(* IEC 61131-3 sources: POMIRTS_lab3/AS/Library_2/AsNxCoM, 3 files *)

(* ---- AsNxCoM.typ ---- *)
TYPE
	nxcomEmcyTelegram_t		: STRUCT			(*emergency telegram*)
		data				: ARRAY[0..7] OF USINT;
	END_STRUCT;

	nxcomEmcyTelegrams_t	: STRUCT			(*array of emergency telegrams*)
		telegram			: ARRAY[0..4] OF nxcomEmcyTelegram_t;
	END_STRUCT;
END_TYPE

(* ---- AsNxCoM.fun ---- *)
{REDUND_CONTEXT} {REDUND_UNREPLICABLE} FUNCTION_BLOCK nxcomGetState			(*get state*)
	VAR_INPUT
		enable			: BOOL;			(*enables execution*)
		pDevice			: UDINT;		(*interface name given as a pointer, e.g., "SL<x>.SS<y>.IF<z>"*)
		node			: USINT;		(*node id*)
		flags			: UDINT;		(*flags*)
	END_VAR
	VAR
        _state			: UINT;			(*internal variable*)
		_result			: UINT;			(*internal variable*)
        _srcId			: UDINT;		(*internal variable*)
	END_VAR
	VAR_OUTPUT
		status			: UINT;			(*execution status: ERR_OK, ERR_FUB_ENABLE_FALSE, ERR_FUB_BUSY, 0xXXXX = see help*)
		coStatus		: UDINT;		(*CANopen stack status*)
		nmtState		: UDINT;		(*state*)
	END_VAR
END_FUNCTION_BLOCK

{REDUND_CONTEXT} {REDUND_UNREPLICABLE} FUNCTION_BLOCK nxcomRecvEmcyDev			(*receive emergency telegrams*)
	VAR_INPUT
		enable			: BOOL;			(*enables execution*)
		pDevice			: UDINT;		(*interface name given as a pointer, e.g., "SL<x>.SS<y>.IF<z>"*)
		node			: USINT;		(*node id*)
		flags			: UDINT;		(*flags*)
		pEmcyData		: UDINT;		(*data field for emergency entries given as pointer (consisting of 5 blocks each sized 8 bytes)*)
	END_VAR
	VAR
        _state			: UINT;			(*internal variable*)
		_result			: UINT;			(*internal variable*)
        _srcId			: UDINT;		(*internal variable*)
	END_VAR
	VAR_OUTPUT
		status			: UINT;			(*execution status: ERR_OK, ERR_FUB_ENABLE_FALSE, ERR_FUB_BUSY, 0xXXXX = see help*)
		coStatus		: UDINT;		(*CANopen stack status*)
		emcyCount		: UDINT;		(*current number of emergency telegrams in buffer*)
	END_VAR
END_FUNCTION_BLOCK

{REDUND_CONTEXT} {REDUND_UNREPLICABLE} FUNCTION_BLOCK nxcomGetDiag				(*get node diagnostics*)
	VAR_INPUT
		enable			: BOOL;			(*enables execution*)
		pDevice			: UDINT;		(*interface name given as a pointer, e.g., "SL<x>.SS<y>.IF<z>"*)
		node			: USINT;		(*node id*)
		flags			: UDINT;		(*flags*)
		pEmcyData		: UDINT;		(*data field for emergency entries given as pointer (consisting of 5 blocks each sized 8 bytes)*)
	END_VAR
	VAR
        _state			: UINT;			(*internal variable*)
		_result			: UINT;			(*internal variable*)
        _srcId			: UDINT;		(*internal variable*)
	END_VAR
	VAR_OUTPUT
		status			: UINT;			(*execution status: ERR_OK, ERR_FUB_ENABLE_FALSE, ERR_FUB_BUSY, 0xXXXX = see help*)
		coStatus		: UDINT;		(*CANopen stack status*)
		nodeFlags		: UDINT;		(*node flags*)
		lastDiagInfo	: UDINT;		(*last diagnostics info*)
		devTypeValid	: BOOL;			(*is device type valid*)
		devType			: UDINT;		(*device type*)
		nmtState		: UDINT;		(*nmt state*)
		emcyCount		: UDINT;		(*current number of emergency telegrams in buffer*)
		addInfo			: UDINT;		(*additional info*)
	END_VAR
END_FUNCTION_BLOCK

{REDUND_CONTEXT} {REDUND_UNREPLICABLE} FUNCTION_BLOCK nxcomNmt					(*send NMT command*)
	VAR_INPUT
		enable			: BOOL;			(*enables execution*)
		pDevice			: UDINT;		(*interface name given as a pointer, e.g., "SL<x>.SS<y>.IF<z>"*)
		node			: USINT;		(*node id*)
		command			: UDINT;		(*NMT command*)
	END_VAR
	VAR
        _state			: UINT;			(*internal variable*)
		_result			: UINT;			(*internal variable*)
        _srcId			: UDINT;		(*internal variable*)
	END_VAR
	VAR_OUTPUT
		status			: UINT;			(*execution status: ERR_OK, ERR_FUB_ENABLE_FALSE, ERR_FUB_BUSY, 0xXXXX = see help*)
		coStatus		: UDINT;		(*CANopen stack status*)
	END_VAR
END_FUNCTION_BLOCK

{REDUND_CONTEXT} {REDUND_UNREPLICABLE} FUNCTION_BLOCK nxcomSdoRead				(*read SDO data*)
	VAR_INPUT
		enable			: BOOL;			(*enables execution*)
		pDevice			: UDINT;		(*interface name given as a pointer, e.g., "SL<x>.SS<y>.IF<z>"*)
		node			: USINT;		(*node id*)
		index			: UDINT;		(*index*)
		subIndex		: UDINT;		(*sub index*)
		dataCount		: UDINT;		(*data count*)
		pData			: UDINT;		(*sdo data given as pointer*)
	END_VAR
	VAR
        _state			: UINT;			(*internal variable*)
		_result			: UINT;			(*internal variable*)
        _srcId			: UDINT;		(*internal variable*)
	END_VAR
	VAR_OUTPUT
		status			: UINT;			(*execution status: ERR_OK, ERR_FUB_ENABLE_FALSE, ERR_FUB_BUSY, 0xXXXX = see help*)
		coStatus		: UDINT;		(*CANopen stack status*)
	END_VAR
END_FUNCTION_BLOCK

{REDUND_CONTEXT} {REDUND_UNREPLICABLE} FUNCTION_BLOCK nxcomSdoWrite			(*write SDO data*)
	VAR_INPUT
		enable			: BOOL;			(*enables execution*)
		pDevice			: UDINT;		(*interface name given as a pointer, e.g., "SL<x>.SS<y>.IF<z>"*)
		node			: USINT;		(*node id*)
		index			: UDINT;		(*index*)
		subIndex		: UDINT;		(*sub index*)
		dataCount		: UDINT;		(*data count*)
		pData			: UDINT;		(*sdo data given as pointer*)
	END_VAR
	VAR
        _state			: UINT;			(*internal variable*)
		_result			: UINT;			(*internal variable*)
        _srcId			: UDINT;		(*internal variable*)
	END_VAR
	VAR_OUTPUT
		status			: UINT;			(*execution status: ERR_OK, ERR_FUB_ENABLE_FALSE, ERR_FUB_BUSY, 0xXXXX = see help*)
		coStatus		: UDINT;		(*CANopen stack status*)
	END_VAR
END_FUNCTION_BLOCK

{REDUND_CONTEXT} {REDUND_UNREPLICABLE} FUNCTION_BLOCK nxcomWriteEmcy			(*write emergency telegrams*)
	VAR_INPUT
		enable			: BOOL;			(*enables execution*)
		pDevice			: UDINT;		(*interface name given as a pointer, e.g., "SL<x>.SS<y>.IF<z>"*)
		errorCode		: UINT;			(*error code*)
		errorRegister	: USINT;		(*error register*)
		pManErrorCode	: UDINT;		(*man error code given as pointer*)
	END_VAR
	VAR
        _state			: UINT;			(*internal variable*)
		_result			: UINT;			(*internal variable*)
        _srcId			: UDINT;		(*internal variable*)
	END_VAR
	VAR_OUTPUT
		status			: UINT;			(*execution status: ERR_OK, ERR_FUB_ENABLE_FALSE, ERR_FUB_BUSY, 0xXXXX = see help*)
		coStatus		: UDINT;		(*CANopen stack status*)
	END_VAR
END_FUNCTION_BLOCK

{REDUND_CONTEXT} {REDUND_UNREPLICABLE} FUNCTION_BLOCK nxcomStartStop			(*start/stop CANopen bus*)
	VAR_INPUT
		enable			: BOOL;			(*enables execution*)
		pDevice			: UDINT;		(*interface name given as a pointer, e.g., "SL<x>.SS<y>.IF<z>"*)
		mode			: UDINT;		(*mode 0 = stop/ 1 = start*)
	END_VAR
	VAR
        _state			: UINT;			(*internal variable*)
		_result			: UINT;			(*internal variable*)
        _srcId			: UDINT;		(*internal variable*)
	END_VAR
	VAR_OUTPUT
		status			: UINT;			(*execution status: ERR_OK, ERR_FUB_ENABLE_FALSE, ERR_FUB_BUSY, 0xXXXX = see help*)
		coStatus		: UDINT;		(*CANopen stack status*)
	END_VAR
END_FUNCTION_BLOCK

{REDUND_CONTEXT} {REDUND_UNREPLICABLE} FUNCTION_BLOCK nxcomSlaveActivate		(*activate/deactivate slave*)
	VAR_INPUT
		enable			: BOOL;			(*enables execution*)
		pDevice			: UDINT;		(*interface name given as a pointer, e.g., "SL<x>.SS<y>.IF<z>"*)
		node			: USINT;		(*node id*)
		mode			: UDINT;		(*mode activate/deactivate slave*)
	END_VAR
	VAR
        _state			: UINT;			(*internal variable*)
		_result			: UINT;			(*internal variable*)
        _srcId			: UDINT;		(*internal variable*)
	END_VAR
	VAR_OUTPUT
		status			: UINT;			(*execution status: ERR_OK, ERR_FUB_ENABLE_FALSE, ERR_FUB_BUSY, 0xXXXX = see help*)
		coStatus		: UDINT;		(*CANopen stack status*)
	END_VAR
END_FUNCTION_BLOCK

(* ---- AsNxCoM.var ---- *)
VAR CONSTANT
	nxcomERR_INVALID_DEVICE					: UINT	:= 34500;		(*error invlaid device*)
	nxcomERR_SEND_MESSAGE					: UINT	:= 34501;		(*error send message*)
	nxcomERR_TIMEOUT						: UINT	:= 34502;		(*error timeout*)
	nxcomERR_CANOPEN_STACK					: UINT	:= 34503;		(*error receive message*)
	nxcomERR_DATALEN						: UINT	:= 34504;		(*error datalen*)
	nxcomERR_PARAMETER						: UINT	:= 34505;		(*error parameter*)

	nxcomNMT_STATE_UNKNOWN					: UDINT	:= 0;			(*unknown*)
	nxcomNMT_STATE_INITIALISING				: UDINT	:= 1;			(*initialising*)
	nxcomNMT_STATE_STOPPED					: UDINT	:= 2;			(*stopped*)
	nxcomNMT_STATE_OPERATIONAL				: UDINT	:= 3;			(*operational*)
	nxcomNMT_STATE_PRE_OPERATIONAL			: UDINT	:= 4;			(*pre-operational*)
	nxcomNMT_STATE_RESET_APPL				: UDINT	:= 5;			(*reset application*)
	nxcomNMT_STATE_RESET_COMM				: UDINT	:= 6;			(*reset communication*)

	nxcomNMT_CMD_START						: UDINT	:= 1;			(*start the node*)
	nxcomNMT_CMD_STOP						: UDINT	:= 2;			(*stop the node*)
	nxcomNMT_CMD_ENTER_PREOP				: UDINT	:= 128;			(*set the node into the pre-operational mode*)
	nxcomNMT_CMD_RESET_NODE					: UDINT	:= 129;			(*reset the node*)
	nxcomNMT_CMD_RESET_COMM					: UDINT	:= 130;			(*reset the communication to the node*)

	nxcomEREG_GENERIC_BIT					: USINT := 16#01;
	nxcomEREG_CURRENT_BIT					: USINT := 16#02;
	nxcomEREG_VOLTAGE_BIT					: USINT := 16#04;
	nxcomEREG_TEMPERATURE_BIT				: USINT := 16#08;
	nxcomEREG_COMM_ERROR_BIT				: USINT := 16#10;
	nxcomEREG_DEV_PROFILE_BIT				: USINT := 16#20;
	nxcomEREG_MANU_SPEC_BIT					: USINT := 16#80;

	nxcomFLAG_PEEK							: UDINT := 16#00000001;	(*node remains in diagnostic lists after request*)

	nxcomNODE_FLAG_DEACTIVATED				: UDINT := 16#80000000; (*node is deactivated and not handled by the master*)
	nxcomNODE_FLAG_STATE_NOT_HANDLED		: UDINT := 16#40000000; (*at least one state has been omitted during the initialization sequence of the node*)
	nxcomNODE_FLAG_INVALID_PARAMETER		: UDINT := 16#00001000; (*parameter set of node is invalid*)
	nxcomNODE_FLAG_UNEXPECTED_BOOTUP		: UDINT := 16#00000800; (*unexpected bootup message from node received*)
	nxcomNODE_FLAG_BOOTUP					: UDINT := 16#00000400; (*expected bootup message from node received*)
	nxcomNODE_FLAG_EMCY_BUFF_OVER			: UDINT := 16#00000200; (*emergency buffer overflow*)
	nxcomNODE_FLAG_EMCY_RECEIVED			: UDINT := 16#00000100; (*emergency telegram received*)
	nxcomNODE_FLAG_UNEXPECTED_STATE			: UDINT := 16#00000080; (*node is in unexpected NMT state*)
	nxcomNODE_FLAG_HEARTBEAT_ERROR			: UDINT := 16#00000040; (*error in heartbeat protocol*)
	nxcomNODE_FLAG_CON_LOST					: UDINT := 16#00000020; (*node guarding has been lost*)
	nxcomNODE_FLAG_GUARD_ERROR				: UDINT := 16#00000010; (*a guarding message has been lost*)
	nxcomNODE_FLAG_HEARTBEAT_STARTED		: UDINT := 16#00000008; (*heartbeat protocol started*)
	nxcomNODE_FLAG_CFG_FAULT				: UDINT := 16#00000004; (*configuration fault*)
	nxcomNODE_FLAG_SDO_ERROR				: UDINT := 16#00000002; (*error during SDO transfer*)
	nxcomNODE_FLAG_SDO_TIMEOUT				: UDINT := 16#00000001; (*timeout during SDO transfer*)

	nxcomMODE_STOP							: UDINT := 0;			(*mode stop*)
	nxcomMODE_START							: UDINT := 1;			(*mode start*)

	nxcomMODE_SLAVE_ACTIVATE				: UDINT := 1;			(*activate slave*)
	nxcomMODE_SLAVE_DEACTIVATE				: UDINT := 2;			(*deactivate slave*)
END_VAR
